TYPE ST_Router_set :
STRUCT
	EnableWifiClient	:	BOOL;
	WifiClientSSID		:	STRING(32) := 'MachineAccessPoint@VDL';
	WifiClientPass		:	STRING(32) := 'e4ff1c12kLL';
	WifiClientSecType	:	eWifiSecurityTypes := eWifiSecurityTypes.PSK2;
	
	EnableWifiAP		:	BOOL;
	WifiAPSSID			:	STRING(32) := 'ePU10_AP';
	WifiAPPass			:	STRING(32) := 'Welkom!VDL';
	WifiAPSecType		:	eWifiSecurityTypes := eWifiSecurityTypes.PSK2;
	
	SimSelectionMode	:	eSimSelectionMode := eSimSelectionMode.auto;
	Sim1Pin				:	STRING(4) := '0000';
	Sim2Pin				:	STRING(4) := '0000';
	
	UpdateSystemTime	:	BOOL;
	
	AutoRebootEnable	:	BOOL;
	ManualReboot		:	BOOL;
END_STRUCT
END_TYPE

(* stored: Version 1.1.0.1, ProductVersion 3.1.4026.18
   DUT ST_Router_set: Id {da4234ff-f25a-4f97-90a2-ae6e9996ae42} *)
